FUNCTION_BLOCK SuspendedToReadyUnifiedProgramTransition EXTENDS SuspendedToReadyProgramTransition
VAR_STAT
	//! <summary>Class name shared by all instances of this function block.</summary>
	{attribute 'OPC.UA.DA' := '0'}
	_ClassName : STRING := __POUNAME();
END_VAR

{attribute 'monitoring' := 'call'}
PROPERTY ClassName : REFERENCE TO STRING
GET
ClassName REF= _ClassName;
END_GET
END_PROPERTY

END_FUNCTION_BLOCK

(* stored: Version 1.1.0.1
   POU SuspendedToReadyUnifiedProgramTransition: Id {b51d8d7c-ce08-44af-83f3-1bc9ae28f472}, SpecialFunc None
   Property ClassName: Id {c4ea174c-042e-4141-88ca-9f33750c28cd}
   Get Get: Id {57b84c67-8afa-4a70-b654-bee3894c192b} *)
